VAR_GLOBAL
	aRxBufferEL			: ARRAY[gc.MINDEVICEINDEX..gc.MAXDEVICEINDEX] OF ComBuffer;	(* Receive data buffer; used with all receive function blocks *)
	aTxBufferEL			: ARRAY[gc.MINDEVICEINDEX..gc.MAXDEVICEINDEX] OF ComBuffer;	(* Transmit data buffer; used with all receive function blocks *)

//	RxBufferKL			: ComBuffer;	(* Receive data buffer; used with all receive function blocks *)
//	TxBufferKL			: ComBuffer;	(* Transmit data buffer; used with all receive function blocks *)
END_VAR

(* stored: Version 1.1.0.1, ProductVersion 3.1.4024.9
   GVL GVL: Id {3e4349e6-a99a-4aa8-b94a-96e30307ccae} *)
